{attribute 'qualified_only'}
{attribute 'to_string'}
TYPE E_TriggerMode :
(
	Off 		:= 0,
	On	 		:= 1
)UDINT;
END_TYPE

(* stored: Version 1.1.0.1, ProductVersion 3.1.4024.13
   DUT E_TriggerMode: Id {5836e03f-3c63-4fdd-a9e8-b007dfce3b03} *)
